// TIA Portal V17 export
// export: Created 2022-01-04T17:38:23.3987438Z, ExportSetting WithDefaults, DisplayName Totally Integrated Automation Portal, DisplayVersion V17, DisplayName TIA Portal Openness, DisplayVersion V17, DisplayName TIA Portal Version Control Interface, DisplayVersion V17, DisplayName STEP 7 Professional, DisplayVersion V17, DisplayName STEP 7 Safety, DisplayVersion V17, DisplayName WinCC Advanced, DisplayVersion V17
DATA_BLOCK "ZadanieFinaloweEKSPERT_DB"   // DB2
VERSION : 0.1
// stored: AutoNumber true, InstanceOfName ZadanieFinaloweEKSPERT, InstanceOfType FB
"ZadanieFinaloweEKSPERT"
   // VAR_INPUT
   //    start : Bool;
   //    stop : Bool;
   //    awaryjneOproznianie : Bool;
   //    czasParzenia : Time;
   //    zadanaIloscWody : Real;
   //    zadanaIloscHerbaty : Real;
   //    temperatura : Int;
   // END_VAR
   // VAR_OUTPUT
   //    przenosnikM1 : Bool;
   //    mieszalnikM2 : Bool;
   //    podgrzewaczG1 : Bool;
   //    otworzZaworZ1 : Bool;
   //    otworzZasuweZ2 : Bool;
   //    otworzZasuweZ3 : Bool;
   //    wodaPoziom : Real;
   //    lisciePoziom : Real;
   //    glownyPoziom : Real;
   // END_VAR
   // VAR
   //    S1 : Bool;
   //    S2 : Bool;
   //    S3 : Bool;
   //    S4 : Bool;
   //    S5 : Bool;
   //    S0 : Bool;
   //    start_edge : Bool;
   //    stop_edge : Bool;
   //    awaryjne_edge : Bool;
   //    S1_Clock : Bool;
   //    w_glownym_wody : Real;
   //    w_glownym_herbaty : Real;
   //    S3_clock : Bool;
   //    M2_edge : Bool;
   //    S5_clock : Bool;
   // END_VAR
BEGIN
END_DATA_BLOCK
